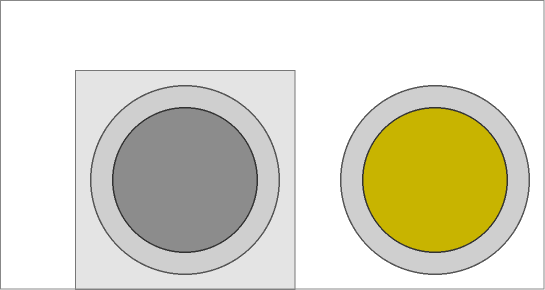
VISUALIZATION Visualization  // 545x290
    PushSwitch (75,70 220x220), variable: IO.HardwareInput[1], behaviour: TAP, style: Switch-PushSwitch-Gray
    Lamp1 (325,70 220x220), variable: IO.HardwareOutput[1], style: Lamp-Lamp1-Yellow
END_VISUALIZATION

(* stored: Version 1.1.0.1, ProductVersion 3.1.4024.12
   Visu Visualization: Id {383a0891-77b0-4ab8-903a-40c998f07fa1} *)
